// Mitsubishi GX Works2 project: plc lab yariv finali   PLC: FX3G

// global labels: Global1
VAR_GLOBAL
  start AT X007 : BOOL;
  analogOutput AT D8282 : INT;
  readyPackages AT D1100 : REAL;
  oatmealInput AT D1110 : REAL;
  oatmealAmount AT D1120 : REAL;
  protein_Input AT D1130 : REAL;
  pwAmount AT D1140 : REAL;
  honeyInput AT D1150 : REAL;
  honeyAmount AT D1160 : REAL;
  missProductAlert AT X005 : BOOL;
  stopAlert AT X005 : BOOL;
  missingProduct AT M0 : BOOL;
  workDay AT Y000 : BOOL;
  productMix AT X003 : BOOL;
  analogInput AT D8280 : INT;
END_VAR
VAR_GLOBAL CONSTANT
  divide : REAL := 400;
  divideNum : REAL := 400;
END_VAR
VAR_GLOBAL
  saveAnalogChoice AT D7000 : REAL;
  pwInput AT D1130 : REAL;
  clasicBar AT D1160 : REAL;
  isClasicBar AT D7000 : REAL;
END_VAR
VAR_GLOBAL CONSTANT
  lowLevelForClasic : REAL := 5;
END_VAR
VAR_GLOBAL
  isProteinBar AT D7000 : REAL;
END_VAR
VAR_GLOBAL CONSTANT
  lowestLevelForProtein : REAL := 5;
END_VAR
VAR_GLOBAL
  clasicSelected AT M5 : BOOL;
  proteinSelected AT M10 : BOOL;
END_VAR
VAR_GLOBAL CONSTANT
  oatmealLowLevelForClasic : REAL := 400;
END_VAR
VAR_GLOBAL
  clasicCheck AT M15 : BOOL;
END_VAR
VAR_GLOBAL CONSTANT
  pwLowLevelForClasic : REAL := 160;
END_VAR
VAR_GLOBAL
  pwClasicCheck AT M20 : BOOL;
  oatmealClasicCheck AT M15 : BOOL;
END_VAR
VAR_GLOBAL CONSTANT
  honeyLowLevelForClasic : REAL := 120;
END_VAR
VAR_GLOBAL
  honeyClasicCheck AT M25 : BOOL;
END_VAR
VAR_GLOBAL CONSTANT
  oatmealLowLevelForProtein : REAL := 240;
END_VAR
VAR_GLOBAL
  oatmealProteinCheck AT M30 : BOOL;
END_VAR
VAR_GLOBAL CONSTANT
  pwLowLevelForProtein : REAL := 320;
END_VAR
VAR_GLOBAL
  pwProteinCheck AT M35 : BOOL;
END_VAR
VAR_GLOBAL CONSTANT
  honeyLowLevelForProtein : REAL := 160;
END_VAR
VAR_GLOBAL
  honeyProteinCheck AT M40 : BOOL;
  clasicAvailable AT M45 : BOOL;
  proteinAvailable AT M50 : BOOL;
END_VAR
VAR_GLOBAL CONSTANT
  isLowerThan5 : REAL := 5;
  isGreaterThan5 : REAL := 5;
  oatmeaForMakeClasic : REAL := 400;
  oatmealNeedForClasic : REAL := 400;
  pwNeedForClasic : REAL := 160;
  honeyNeedForClasic : REAL := 120;
  oatmealNeedForProtein : REAL := 240;
  pwNeedForProtein : REAL := 320;
  honeyNeedForProtein : REAL := 160;
END_VAR
VAR_GLOBAL
  mixTime AT Y003 : BOOL;
  y3Light AT TS0 : BOOL;
END_VAR
VAR_GLOBAL CONSTANT
  mixingTime : INT := 50;
END_VAR
VAR_GLOBAL
  y3Lighting AT TC0 : BOOL;
  oven AT D1170 : REAL;
END_VAR
VAR_GLOBAL CONSTANT
  clasicIngredients : REAL := 680;
  proteinIngredients : REAL := 720;
  clasicBaking : REAL := 1;
  proteinBaking : REAL := 1;
END_VAR
VAR_GLOBAL
  clasicBake AT D1170 : REAL;
  proteinBake AT D1180 : REAL;
  timeToBake AT TS0 : BOOL;
  readyToBake AT M55 : BOOL;
  startBake AT X002 : BOOL;
  y_5 AT Y005 : BOOL;
  y_6 AT Y006 : BOOL;
  M_0 : BOOL;
  ts_5 AT TS5 : BOOL;
  ts_6 AT TS6 : BOOL;
  M_1 : BOOL;
  M_60 AT M60 : BOOL;
  M_65 AT M65 : BOOL;
  y_1 AT Y001 : BOOL;
  y_2 AT Y002 : BOOL;
  ts_1 AT TS1 : BOOL;
  ts_2 AT TS2 : BOOL;
  tc_1 AT TC1 : BOOL;
  tc_2 AT TC2 : BOOL;
END_VAR
VAR_GLOBAL CONSTANT
  blink_time : INT := 5;
  blink_time2 : INT := 10;
END_VAR
VAR_GLOBAL
  tx_1 AT TC2 : BOOL;
END_VAR
VAR_GLOBAL CONSTANT
  TC1 : INT := 10;
END_VAR
VAR_GLOBAL
  tc_5 AT TC5 : BOOL;
  classic_mix_time AT TC5 : BOOL;
END_VAR
VAR_GLOBAL CONSTANT
  classicMixTime : INT := 40;
END_VAR
VAR_GLOBAL
  tc_4 AT TC4 : BOOL;
END_VAR
VAR_GLOBAL CONSTANT
  protainMixTime : INT := 50;
END_VAR
VAR_GLOBAL
  start_packing AT X006 : BOOL;
  cc1 AT CC1 : BOOL;
  one_unit_packing AT X000 : BOOL;
END_VAR
VAR_GLOBAL CONSTANT
  oneSnack : INT := 1;
END_VAR
VAR_GLOBAL
  cc2 AT CC2 : BOOL;
END_VAR
VAR_GLOBAL CONSTANT
  seven_gumigum : INT := 8;
END_VAR
VAR_GLOBAL
  cs1 AT CS1 : BOOL;
  lastOnePack AT CS2 : BOOL;
  packing_in_process AT Y004 : BOOL;
  packing_end AT M11 : BOOL;
  reset_counters AT X007 : BOOL;
  one_unit_start AT CC1 : BOOL;
  full_pack AT CC2 : BOOL;
  ready_packs AT D1100 : REAL;
END_VAR
VAR_GLOBAL CONSTANT
  add_1 : REAL := 1;
END_VAR
VAR_GLOBAL
  M_166 AT M166 : BOOL;
END_VAR

// task Task_01 (event TRUE, interval 0, priority 31): POU_01

PROGRAM POU_01
VAR
  proteinInput : REAL;
  product_Mix : REAL;
  produc_tMix : REAL;
  M_26 : BOOL;
END_VAR
(* structured ladder/FBD written out as ST: instructions are called as NAME(EN, inputs, outputs); _pN, _eN, _tN stand for wires *)
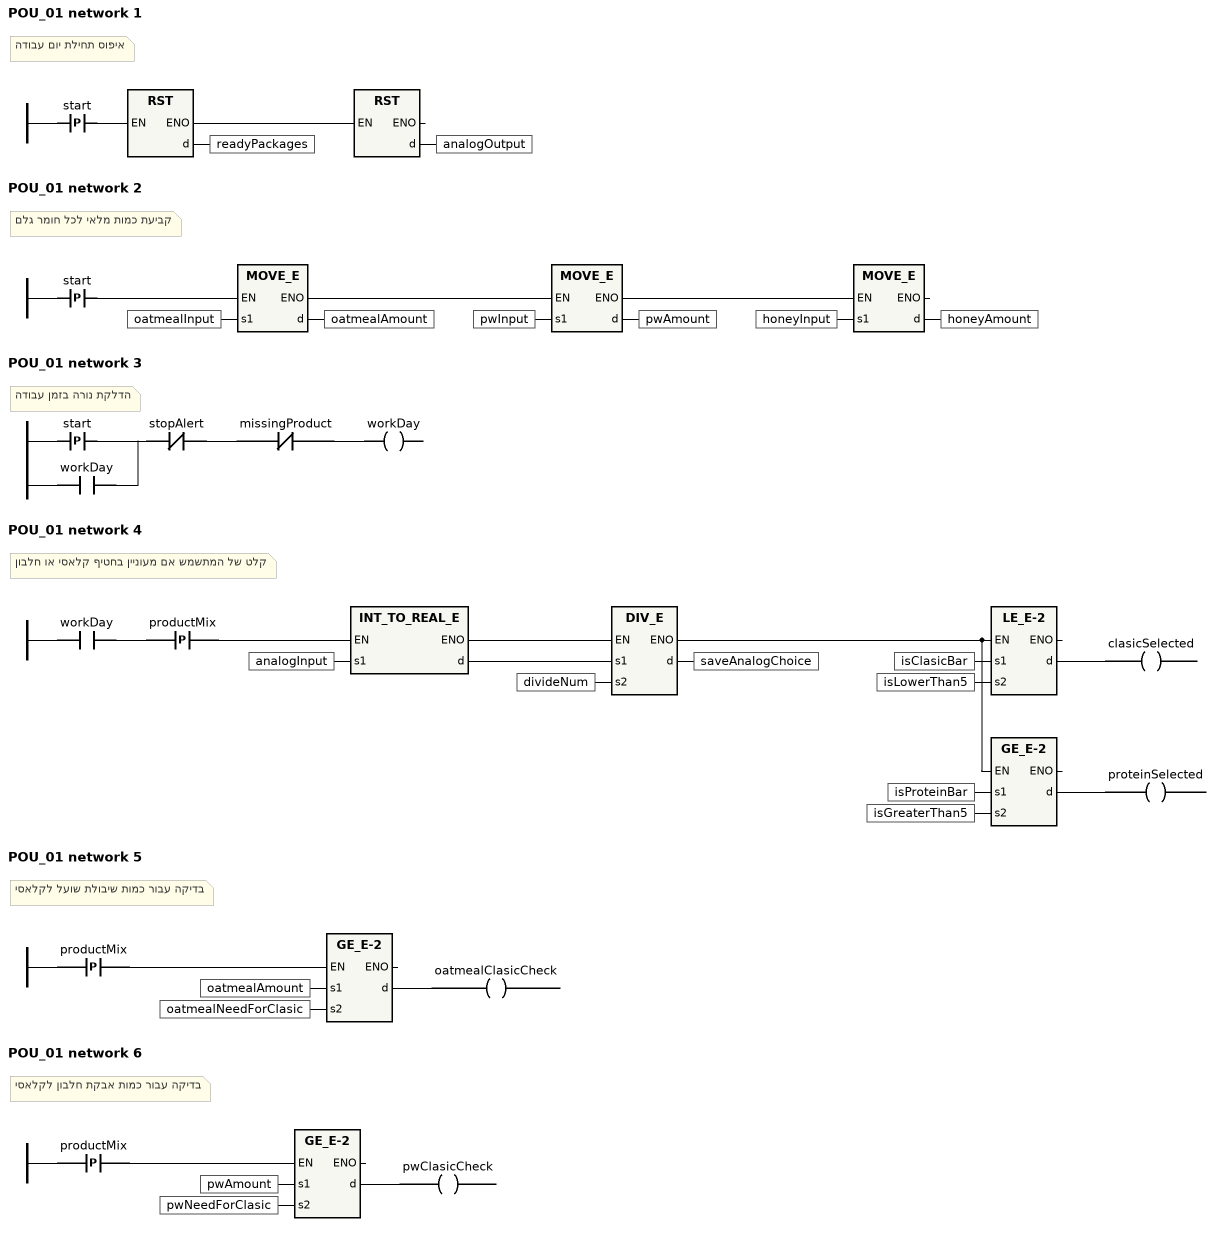
(* network 1 *)
(* איפוס תחילת יום עבודה *)
_e1 := RST(LDP(TRUE, start), readyPackages);
RST(_e1, analogOutput);
(* network 2 *)
(* קביעת כמות מלאי לכל חומר גלם *)
_e1 := MOVE_E(LDP(TRUE, start), oatmealInput, oatmealAmount);
_e2 := MOVE_E(_e1, pwInput, pwAmount);
MOVE_E(_e2, honeyInput, honeyAmount);
(* network 3 *)
(* הדלקת נורה בזמן עבודה *)
workDay := ((LDP(TRUE, start) OR workDay) AND NOT stopAlert) AND NOT missingProduct;
(* network 4 *)
(* קלט של המתשמש אם מעוניין בחטיף קלאסי או חלבון *)
_e2 := INT_TO_REAL_E(workDay AND LDP(TRUE, productMix), analogInput, _t1);
_e3 := DIV_E(_e2, _t1, divideNum, saveAnalogChoice);
LE_E(_e3, isClasicBar, isLowerThan5, _t4);
clasicSelected := _t4;
GE_E(_e3, isProteinBar, isGreaterThan5, _t5);
proteinSelected := _t5;
(* network 5 *)
(* בדיקה עבור כמות שיבולת שועל לקלאסי *)
GE_E(LDP(TRUE, productMix), oatmealAmount, oatmealNeedForClasic, _t1);
oatmealClasicCheck := _t1;
(* network 6 *)
(* בדיקה עבור כמות אבקת חלבון לקלאסי *)
GE_E(LDP(TRUE, productMix), pwAmount, pwNeedForClasic, _t1);
pwClasicCheck := _t1;
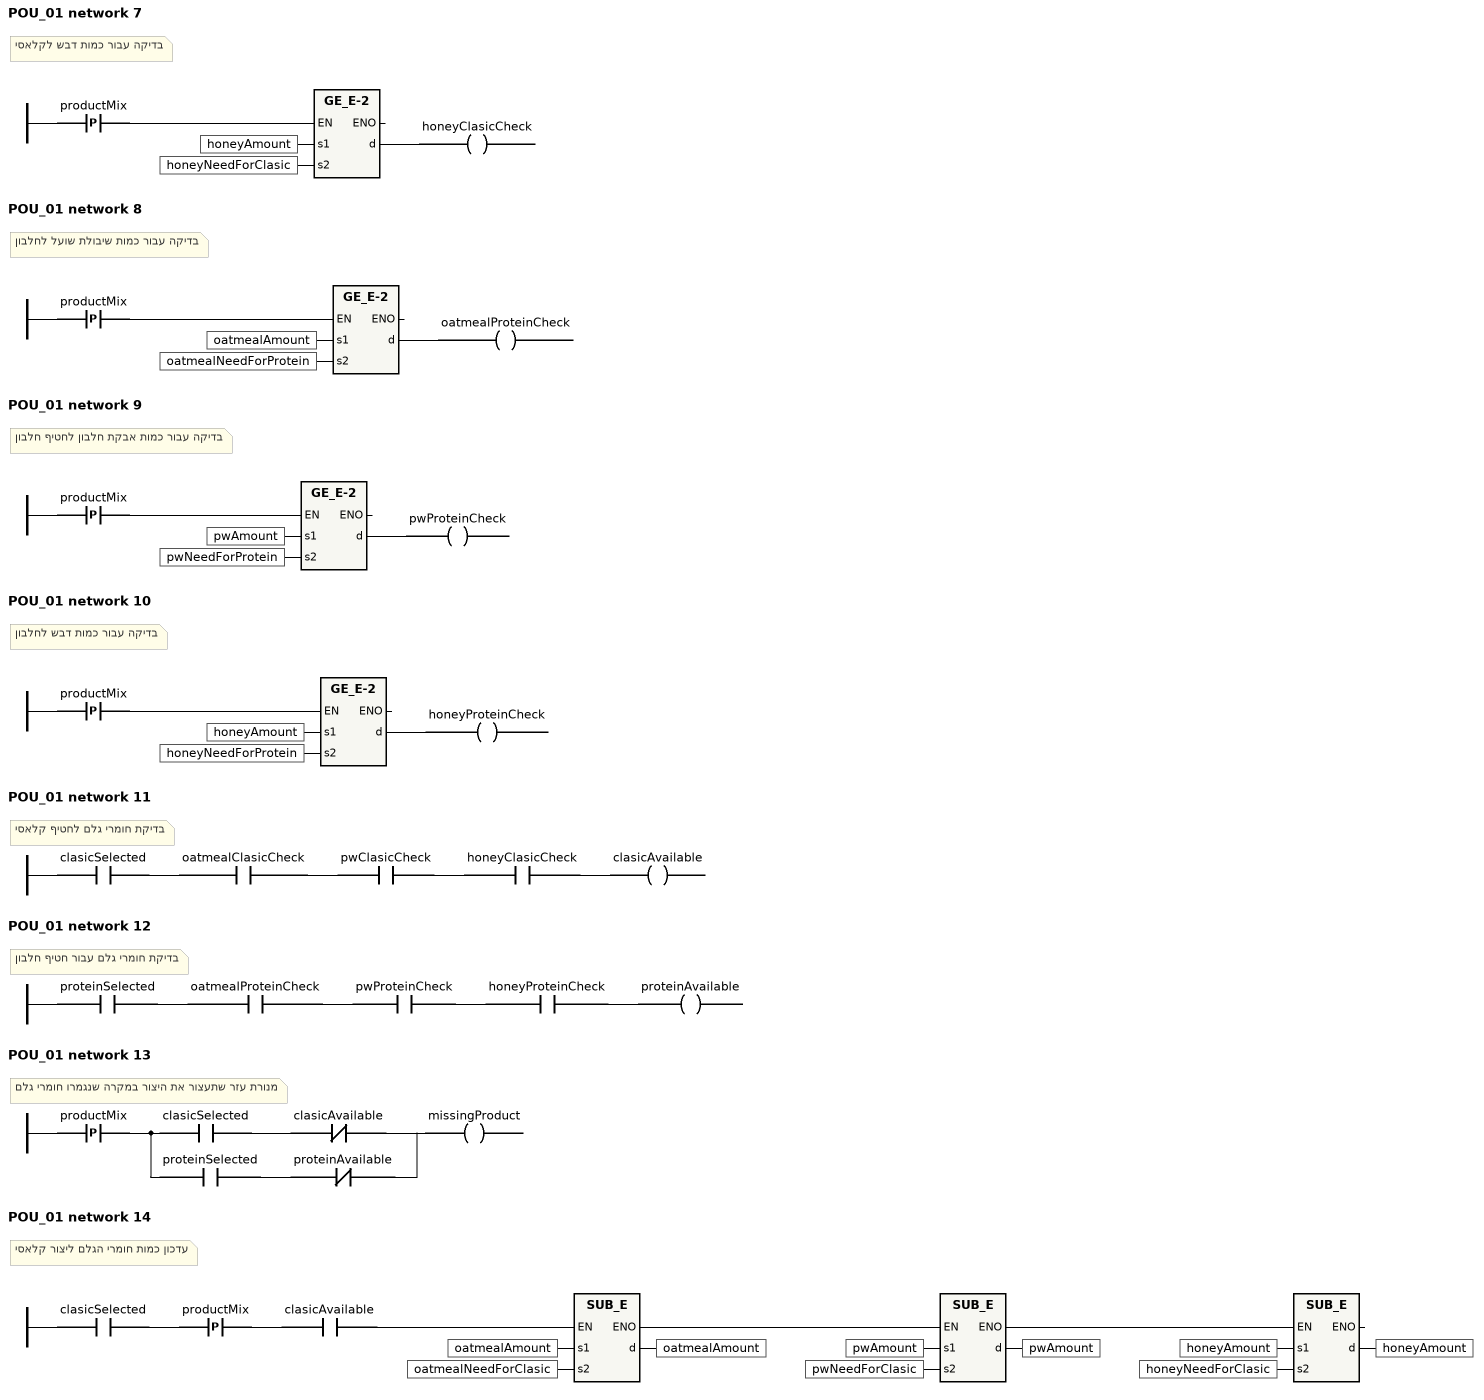
(* network 7 *)
(* בדיקה עבור כמות דבש לקלאסי *)
GE_E(LDP(TRUE, productMix), honeyAmount, honeyNeedForClasic, _t1);
honeyClasicCheck := _t1;
(* network 8 *)
(* בדיקה עבור כמות שיבולת שועל לחלבון *)
GE_E(LDP(TRUE, productMix), oatmealAmount, oatmealNeedForProtein, _t1);
oatmealProteinCheck := _t1;
(* network 9 *)
(* בדיקה עבור כמות אבקת חלבון לחטיף חלבון *)
GE_E(LDP(TRUE, productMix), pwAmount, pwNeedForProtein, _t1);
pwProteinCheck := _t1;
(* network 10 *)
(* בדיקה עבור כמות דבש לחלבון *)
GE_E(LDP(TRUE, productMix), honeyAmount, honeyNeedForProtein, _t1);
honeyProteinCheck := _t1;
(* network 11 *)
(* בדיקת חומרי גלם לחטיף קלאסי *)
clasicAvailable := clasicSelected AND oatmealClasicCheck AND pwClasicCheck AND honeyClasicCheck;
(* network 12 *)
(* בדיקת חומרי גלם עבור חטיף חלבון *)
proteinAvailable := proteinSelected AND oatmealProteinCheck AND pwProteinCheck AND honeyProteinCheck;
(* network 13 *)
(* מנורת עזר שתעצור את היצור במקרה שנגמרו חומרי גלם *)
_p1 := LDP(TRUE, productMix);
missingProduct := (_p1 AND clasicSelected AND NOT clasicAvailable) OR (_p1 AND proteinSelected AND NOT proteinAvailable);
(* network 14 *)
(* עדכון כמות חומרי הגלם ליצור קלאסי *)
_e1 := SUB_E(clasicSelected AND LDP(TRUE, productMix) AND clasicAvailable, oatmealAmount, oatmealNeedForClasic, oatmealAmount);
_e2 := SUB_E(_e1, pwAmount, pwNeedForClasic, pwAmount);
SUB_E(_e2, honeyAmount, honeyNeedForClasic, honeyAmount);
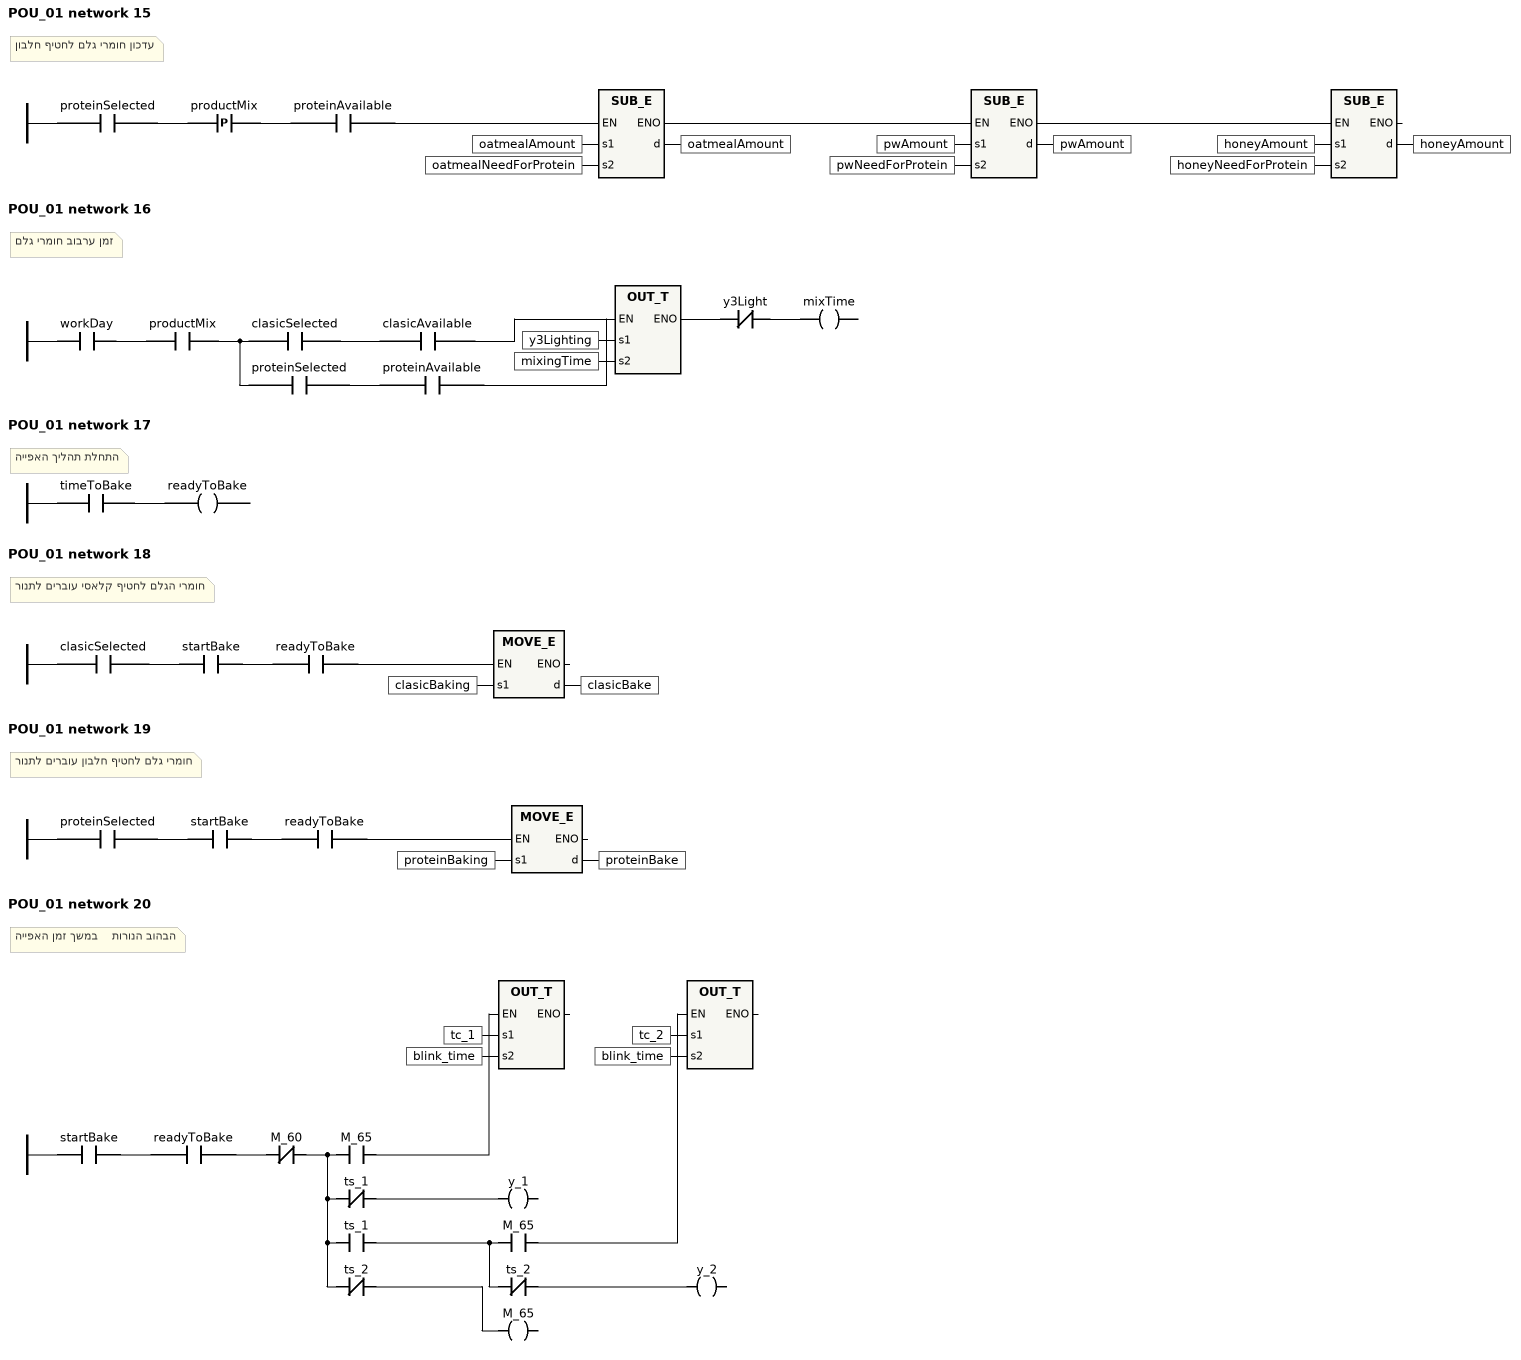
(* network 15 *)
(* עדכון חומרי גלם לחטיף חלבון *)
_e1 := SUB_E(proteinSelected AND LDP(TRUE, productMix) AND proteinAvailable, oatmealAmount, oatmealNeedForProtein, oatmealAmount);
_e2 := SUB_E(_e1, pwAmount, pwNeedForProtein, pwAmount);
SUB_E(_e2, honeyAmount, honeyNeedForProtein, honeyAmount);
(* network 16 *)
(* זמן ערבוב חומרי גלם *)
_p1 := workDay AND productMix;
_e2 := OUT_T((_p1 AND clasicSelected AND clasicAvailable) OR (_p1 AND proteinSelected AND proteinAvailable), y3Lighting, mixingTime);
mixTime := _e2 AND NOT y3Light;
(* network 17 *)
(* התחלת תהליך האפייה *)
readyToBake := timeToBake;
(* network 18 *)
(* חומרי הגלם לחטיף קלאסי עוברים לתנור *)
MOVE_E(clasicSelected AND startBake AND readyToBake, clasicBaking, clasicBake);
(* network 19 *)
(* חומרי גלם לחטיף חלבון עוברים לתנור *)
MOVE_E(proteinSelected AND startBake AND readyToBake, proteinBaking, proteinBake);
(* network 20 *)
(* הבהוב הנורות    במשך זמן האפייה *)
_p1 := startBake AND readyToBake AND NOT M_60;
OUT_T(_p1 AND M_65, tc_1, blink_time);
y_1 := _p1 AND NOT ts_1;
_p2 := _p1 AND ts_1;
OUT_T(_p2 AND M_65, tc_2, blink_time);
y_2 := _p2 AND NOT ts_2;
M_65 := _p1 AND NOT ts_2;
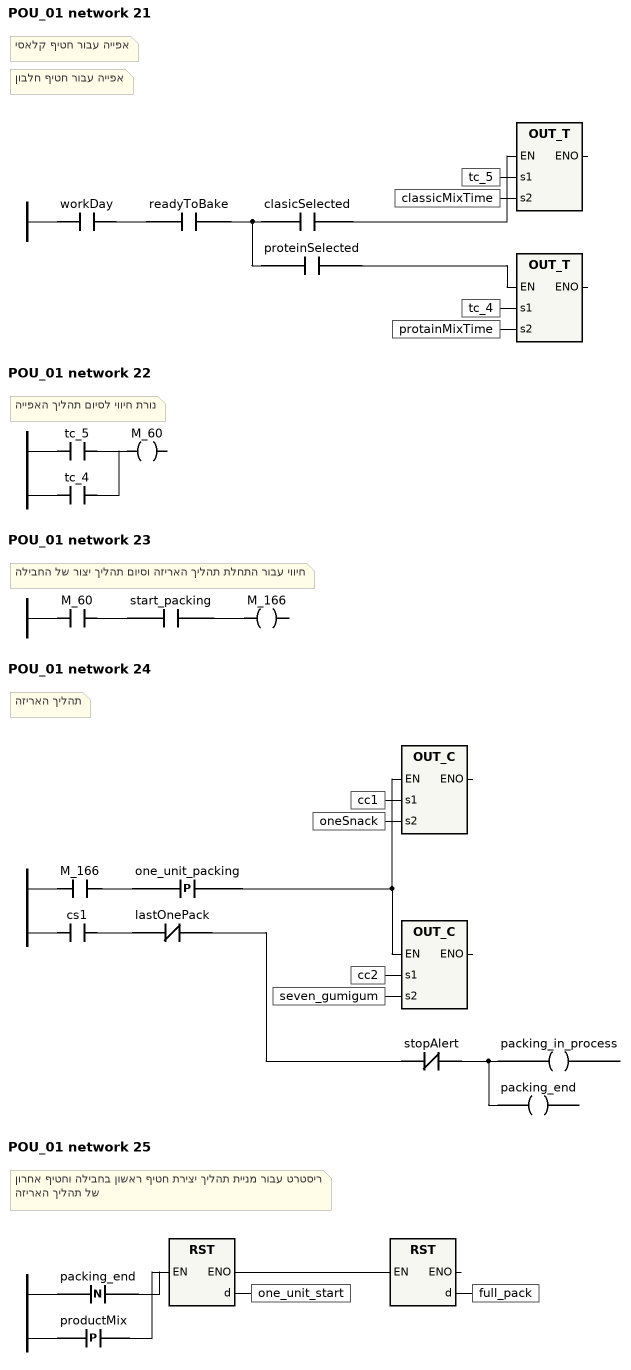
(* network 21 *)
(* אפייה עבור חטיף קלאסי *)
(* אפייה עבור חטיף חלבון *)
_p1 := workDay AND readyToBake;
OUT_T(_p1 AND clasicSelected, tc_5, classicMixTime);
OUT_T(_p1 AND proteinSelected, tc_4, protainMixTime);
(* network 22 *)
(* נורת חיווי לסיום תהליך האפייה *)
M_60 := tc_5 OR tc_4;
(* network 23 *)
(* חיווי עבור התחלת תהליך האריזה וסיום תהליך יצור של החבילה *)
M_166 := M_60 AND start_packing;
(* network 24 *)
(* תהליך האריזה *)
_p1 := M_166 AND LDP(TRUE, one_unit_packing);
OUT_C(_p1, cc1, oneSnack);
OUT_C(_p1, cc2, seven_gumigum);
_p2 := cs1 AND NOT lastOnePack AND NOT stopAlert;
packing_in_process := _p2;
packing_end := _p2;
(* network 25 *)
(* ריסטרט עבור מניית תהליך יצירת חטיף ראשון בחבילה וחטיף אחרון של תהליך האריזה *)
_e1 := RST(LDF(TRUE, packing_end) OR LDP(TRUE, productMix), one_unit_start);
RST(_e1, full_pack);
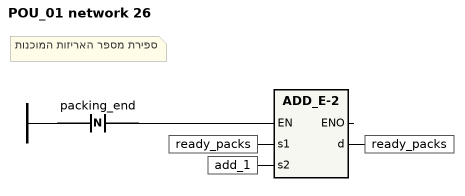
(* network 26 *)
(* ספירת מספר האריזות המוכנות *)
ADD_E(LDF(TRUE, packing_end), ready_packs, add_1, ready_packs);
END_PROGRAM
